FUNCTION_BLOCK FB_SmoothAxis
VAR_INPUT
	i_xHotPlug	:	BOOL;
END_VAR
VAR_OUTPUT
	q_asResult: ARRAY [1..20] OF STRING;
	q_xError	:	BOOL;
END_VAR
VAR_IN_OUT
	iq_Axis	:	ST_HOMSStepper;
END_VAR
VAR

	mcPower	:	MC_Power;
	mcReset	:	MC_Reset;
	mcMoveAbsolute : ARRAY[1..2] OF MC_MoveAbsolute;
	mcHalt	:	MC_Halt;
	mcSmoothMover	:	MC_SmoothMover;
	//Error Stuff
	indexResult: INT := 1;
	fbFormatString	:	FB_FormatString;
	
	xInitComplete	:	BOOL := FALSE;
	
	imcBlockIndex: INT;
	
	rtEnable : R_TRIG;
	ftEnable : F_TRIG;
	rtStop	:	R_TRIG;
	rtStart	:	R_TRIG;
	rReqAbsPosOld: REAL := 0;
	rReqAbsPosPrevious: REAL;
	iI: INT;
END_VAR

(* Manipulator Axis Function Block
Alex Wallace, 2016-8-8 

This block works by jumping between two absolute move blocks and buffering
the motion between them.
*)


rtEnable(CLK:=iq_Axis.xEnable);
ftEnable(CLK:=iq_Axis.xEnable);

//Update status
iq_Axis.stAxis();

IF rtEnable.Q OR ftEnable.Q THEN
	xInitComplete := FALSE;
	iq_Axis.eState := Init;
ELSIF xInitComplete THEN
	iq_Axis.eState := MoveEnabled;
END_IF

//For EPICS, because the modbus map was made for 32 bit..
iq_Axis.rActPos := LREAL_TO_REAL(iq_Axis.stAxis.NcToPlc.ActPos);


CASE iq_Axis.eState OF
	0: iq_Axis.eState := Init;
	Init:
	(* Start by initializing the motor axis *)
	mcPower.Enable := iq_Axis.xEnable;
	iq_Axis.rReqAbsPos := iq_Axis.rActPos; //do this when the PLC comes up so we don't just lose the position if we tweak
	IF mcPower.Status THEN //success
		xInitComplete := TRUE;
		q_asResult[indexResult] := 'Motor init success';
		indexResult := indexResult + 1;
		iq_Axis.eState := MoveEnabled;
	ELSIF mcPower.Error THEN
		mcPower.Enable := FALSE;
		fbFormatString(sFormat:='Init mcPower Error: %s', arg1:=F_UDINT(mcPower.ErrorID));
		ActError();
	END_IF
		
	MoveEnabled:
		mcSmoothMover.Enable := iq_Axis.xEnable;
		mcSmoothMover.ReqAbsPos := LIMIT(-100, REAL_TO_LREAL(iq_Axis.rReqAbsolute), 100);
		mcSmoothMover.Execute := iq_Axis.xStart;
		(*We've already captured the rising edge of start (if there was one, so 
		go ahead and reset it.*)
		iq_Axis.xStart := FALSE;
		
		//Halt
		mcHalt.Execute S= iq_Axis.xStop;
		mcHalt.Execute R= mcHalt.Busy;
		iq_Axis.xStop R= mcHalt.Busy;
		IF mcPower.Error OR mcSmoothMover.Error THEN
			iq_Axis.eState:=Error;
		END_IF
		
	Error:
		mcReset.Execute := rtEnable.Q OR i_xHotPlug OR iq_Axis.xReset;
		IF mcReset.Done THEN
			q_xError := FALSE;
			mcReset.Execute := FALSE;
			iq_Axis.xReset := FALSE;
			iq_Axis.eState:=Init;
		END_IF
	
END_CASE


(* Run the mc blocks *)
ActPower();
mcReset(Axis:=iq_Axis.stAxis);
mcSmoothMover(Axis:=iq_Axis.stAxis,
	Velocity:=iq_Axis.fVelocity);
mcHalt(Axis:=iq_Axis.stAxis);

iq_Axis.bDone := mcHalt.Done OR mcSmoothMover.Done;
iq_Axis.bBusy := mcHalt.Busy OR mcSmoothMover.Busy;

//For display, this logic is not for safety
iq_Axis.xHiLS := NOT iq_Axis.xHiLS;
iq_Axis.xLoLS := NOT iq_Axis.xLoLS;

ACTION ActError:
(* Error action
*)

//Reset the debugging index
IF indexResult > 20 THEN indexResult := 1; END_IF

iq_Axis.eState := Error;
q_xError	:=	TRUE;
q_asResult[indexResult] := fbFormatString.sOut;
indexResult := indexResult +1;
END_ACTION

ACTION ActPower:
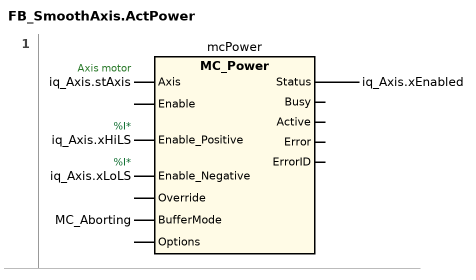
// NETWORK 1
//   iq_Axis.stAxis: Axis motor
//   iq_Axis.xHiLS: AT %I*
//   iq_Axis.xLoLS: AT %I*
mcPower(
    Axis := iq_Axis.stAxis,
    Enable_Positive := iq_Axis.xHiLS,
    Enable_Negative := iq_Axis.xLoLS,
    BufferMode := MC_Aborting); // MC_Power
iq_Axis.xEnabled := mcPower.Status;
END_ACTION

END_FUNCTION_BLOCK

(* stored: Version 1.1.0.1, ProductVersion 3.1.4020.12
   POU FB_SmoothAxis: Id {2c576ec6-7433-4ec0-8547-ab9b5dd393c9}, SpecialFunc None
   Action ActError: Id {efb14a67-3fcd-4d5f-a82f-60b8d6779b53}
   Action ActPower: Id {31b74a81-1b68-4db8-b9a3-64793fff0f5a} *)
